{attribute 'GeneratedUsingTerminal: EK1122-0000-0018'}
{attribute addProperty BoxType "EK1122-0000-0018"}
{attribute addProperty Id "Beckhoff_EJ7xxxsub_EK1100EK1100_1FC0878B2"}
{attribute addProperty CRC "977515042"}
{attribute addProperty Size "2"}
{attribute addProperty Name "Beckhoff EJ7xxxEK1122"}
TYPE Beckhoff_EJ7xxxEK1122_3A43B222 EXTENDS EK1122_1FC0878B :
STRUCT
	{attribute addProperty Name "Beckhoff EJ7xxxsub EK1100"}
	{attribute addProperty PreviousPort "Beckhoff EJ7xxxEK1122 : D"}
	Beckhoff_EJ7xxxsub_EK1100 : EK1100_1FC0878B;
END_STRUCT
END_TYPE

(* stored: Version 1.2.0.0, ProductVersion 3.1.4024.11
   DUT Beckhoff_EJ7xxxEK1122_3A43B222: Id {bd5516ea-4fb6-4d1c-9406-e245fdf87c08} *)
